// TIA Portal V15.1 export
// export: Created 2026-01-09T13:45:12.180441Z, ExportSetting WithDefaults, WithReadOnly, DisplayName Totally Integrated Automation Portal, DisplayVersion V15.1 Update 8, DisplayName TIA Portal Openness, DisplayVersion V15.1 Update 8, DisplayName STEP 7 Professional, DisplayVersion V15.1 Update 8, DisplayName WinCC Advanced, DisplayVersion V15.1 Update 8
FUNCTION "2.MOVE_OUT" : Void   // FC2, LAD
{ S7_Optimized_Access := 'TRUE' }
VERSION : 0.1
// stored: AutoNumber false, CodeModifiedDate 2025-08-27T17:06:54.9207011Z, CompileDate 2025-08-30T17:40:33.361501Z, CreationDate 2024-10-12T12:36:08.0193576Z, HandleErrorsWithinBlock false, InterfaceModifiedDate 2023-08-09T15:10:11.0888586Z, IsConsistent true, IsIECCheckEnabled false, IsKnowHowProtected false, IsWriteProtected false, LibraryConformanceStatus The object is library-conformant., ModifiedDate 2025-08-27T17:06:54.9207011Z, ParameterModified 2023-08-09T15:10:11.0888586Z, PLCSimAdvancedSupport false, SetENOAutomatically False, StructureModified 2023-08-09T15:10:11.0888586Z, UDAEnableTagReadback false
   VAR_INPUT
      "0.0" : Bool;
      "0.1" : Bool;
      "0.2" : Bool;
      "0.3" : Bool;
      "0.4" : Bool;
      "0.5" : Bool;
      "0.6" : Bool;
      "0.7" : Bool;
   END_VAR
   VAR_OUTPUT
      "0_0" : Bool;
      "0_1" : Bool;
      "0_2" : Bool;
      "0_3" : Bool;
      "0_4" : Bool;
      "0_5" : Bool;
      "0_6" : Bool;
      "0_7" : Bool;
   END_VAR
BEGIN

REGION Network 3
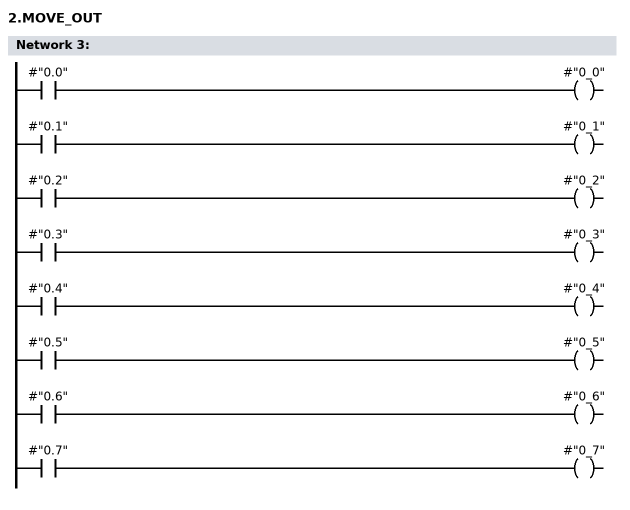
   RUNG wire#powerrail
      Contact( #"0.0" )
      Coil( #"0_0" )
   END_RUNG
   RUNG wire#powerrail
      Contact( #"0.1" )
      Coil( #"0_1" )
   END_RUNG
   RUNG wire#powerrail
      Contact( #"0.2" )
      Coil( #"0_2" )
   END_RUNG
   RUNG wire#powerrail
      Contact( #"0.3" )
      Coil( #"0_3" )
   END_RUNG
   RUNG wire#powerrail
      Contact( #"0.4" )
      Coil( #"0_4" )
   END_RUNG
   RUNG wire#powerrail
      Contact( #"0.5" )
      Coil( #"0_5" )
   END_RUNG
   RUNG wire#powerrail
      Contact( #"0.6" )
      Coil( #"0_6" )
   END_RUNG
   RUNG wire#powerrail
      Contact( #"0.7" )
      Coil( #"0_7" )
   END_RUNG
   // the same network as SCL:
   #"0_0" := #"0.0";
   #"0_1" := #"0.1";
   #"0_2" := #"0.2";
   #"0_3" := #"0.3";
   #"0_4" := #"0.4";
   #"0_5" := #"0.5";
   #"0_6" := #"0.6";
   #"0_7" := #"0.7";
END_REGION
END_FUNCTION
